# EPICS StreamDevice protocol: ldens3300Sup/ldens3300.proto
InTerminator = CR LF;

getTemperature {
    in "T= %f %*s D= %*f %*s";
}

getDensity {
    in "T= %*f %*s D= %f %*s";
}
